INTERFACE I_MoveVelo

PROPERTY Acceleration : MC_LREAL
GET
END_GET
SET
END_SET
END_PROPERTY

PROPERTY BufferMode : MC_Buffermode
GET
END_GET
SET
END_SET
END_PROPERTY

PROPERTY Busy : BOOL
GET
END_GET
END_PROPERTY

PROPERTY Deceleration : MC_LREAL
GET
END_GET
SET
END_SET
END_PROPERTY

PROPERTY Direction : MC_Direction
GET
END_GET
SET
END_SET
END_PROPERTY

PROPERTY Error : BOOL
GET
END_GET
END_PROPERTY

PROPERTY Execute : BOOL
GET
END_GET
SET
END_SET
END_PROPERTY

PROPERTY InVelocity : BOOL
GET
END_GET
END_PROPERTY

PROPERTY Jerk : MC_LREAL
GET
END_GET
SET
END_SET
END_PROPERTY

PROPERTY Velocity : MC_LREAL
GET
END_GET
SET
END_SET
END_PROPERTY

END_INTERFACE

(* stored: Version 1.1.0.1
   Itf I_MoveVelo: Id {ee1ce8a7-ec58-44d9-b1cd-a5a424d1d3e4}
   Property Acceleration: Id {7ccc0940-958c-495e-8503-eece6a8b4378}
   Get Get: Id {43d91512-0933-43fc-959b-33b47cac4760}
   Set Set: Id {44887457-45f1-4fd0-938d-269a4c0a2129}
   Property BufferMode: Id {b4bd8e46-17f0-4dd2-9baa-56ba1d2a6fff}
   Get Get: Id {2a790a3e-3257-40aa-9193-707c9086b013}
   Set Set: Id {1005d255-5562-4c61-9919-30043be82e3f}
   Property Busy: Id {933b7b25-55f7-499a-92cd-f00162f79c82}
   Get Get: Id {8fafce60-2b89-4caa-a433-5672c80f58b3}
   Property Deceleration: Id {fc33ab26-668b-4c72-a709-23a15799cca0}
   Get Get: Id {90ba0b5c-dbee-40a7-bb9f-7ce884114315}
   Set Set: Id {cb7b807e-6fdb-4f54-aa34-ff4c3d0ca38b}
   Property Direction: Id {489282e3-22b2-46a5-9130-7dda39eb73b1}
   Get Get: Id {dad66055-30bd-44f4-8a19-aeda29e72a83}
   Set Set: Id {b58701bb-56d0-4907-b495-9b810b1129ac}
   Property Error: Id {f8823bc0-59f3-4afa-8bac-650825464243}
   Get Get: Id {42f9a81b-ebe2-43cc-b0a9-28bf984ea94e}
   Property Execute: Id {9f2791c4-54a4-46d7-a104-098b5be21111}
   Get Get: Id {8330fc1f-33f5-480e-a46b-84d9bf522542}
   Set Set: Id {4637af2c-dca8-45dc-9000-6cb308af81cc}
   Property InVelocity: Id {39525ada-6c93-4893-94d3-28de654c4cfd}
   Get Get: Id {6f0cdd5e-8420-41f0-9dee-ed50de3ee874}
   Property Jerk: Id {08472ee4-cdc9-43cd-9e3d-4dee835a41f7}
   Get Get: Id {60c3ac36-fd7a-43ea-ac00-7d87094497f5}
   Set Set: Id {2aa45ff3-8d50-4fdf-8fc9-463458ff8a64}
   Property Velocity: Id {a66b21b9-2298-460e-a241-527c14218e5c}
   Get Get: Id {a85af41f-39f4-41a2-b765-639388cca9e7}
   Set Set: Id {2eec48cd-d3e6-493f-95fa-f598f9ca3b3a} *)
